FUNCTION FC_BroachingPlanCopyPass
VAR_INPUT
	pByte : POINTER TO BYTE;
	BaseBroachingPlan 		: DUT_stBroachingPlanBase;     
    VariantsBroachingPlan	: DUT_stBroachingPlanVariants;
END_VAR

pByte[0]	:= DINT_TO_BYTE(BaseBroachingPlan.ToolHolderBase_Position);
pByte[1]	:= DINT_TO_BYTE(VariantsBroachingPlan.ToolHolderA_Position);
pByte[2]	:= DINT_TO_BYTE(VariantsBroachingPlan.ToolHolderB_Position);
pByte[3]	:= DINT_TO_BYTE(VariantsBroachingPlan.ToolHolderC_Position);
pByte[4]	:= DINT_TO_BYTE(VariantsBroachingPlan.ToolHolderD_Position);
pByte[5] 	:= DINT_TO_BYTE(VariantsBroachingPlan.ToolHolderE_Position);
pByte[6] 	:= DINT_TO_BYTE(VariantsBroachingPlan.ToolHolderF_Position);

END_FUNCTION

(* stored: Version 1.1.0.1, ProductVersion 3.1.4024.15
   POU FC_BroachingPlanCopyPass: Id {e2e1860e-d379-4368-9322-033e6802402c}, SpecialFunc None *)
